FUNCTION_BLOCK SS5b_ps_Ejector (* Composite FB wrapping other FBs *)
  (* Standard: 61499-2 *)
  (* Version 1.0, 2025-08-26, PS_Transformer_for_Unknown *)
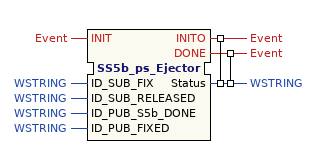
  EVENT_INPUT
    INIT; (* Initialization Request *)
  END_EVENT
  EVENT_OUTPUT
    INITO WITH Status; (* Initialization Confirm *)
    DONE WITH Status; (* Execution Confirmation *)
  END_EVENT
  VAR_INPUT
    ID_SUB_FIX : WSTRING;
    ID_SUB_RELEASED : WSTRING;
    ID_PUB_S5b_DONE : WSTRING;
    ID_PUB_FIXED : WSTRING;
  END_VAR
  VAR_OUTPUT
    Status : WSTRING; (* Output event qualifier *)
  END_VAR
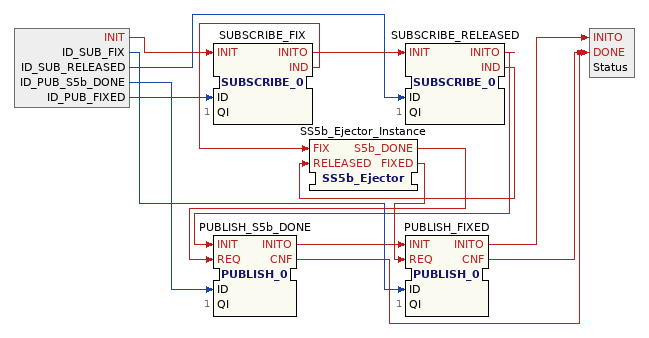
  FBS
    SS5b_Ejector_Instance : SS5b_Ejector;
    SUBSCRIBE_FIX : SUBSCRIBE_0(QI := 1);
    SUBSCRIBE_RELEASED : SUBSCRIBE_0(QI := 1);
    PUBLISH_S5b_DONE : PUBLISH_0(QI := 1);
    PUBLISH_FIXED : PUBLISH_0(QI := 1);
  END_FBS
  EVENT_CONNECTIONS
    INIT TO SUBSCRIBE_FIX.INIT;
    SUBSCRIBE_FIX.INITO TO SUBSCRIBE_RELEASED.INIT;
    SUBSCRIBE_RELEASED.INITO TO PUBLISH_S5b_DONE.INIT;
    PUBLISH_S5b_DONE.INITO TO PUBLISH_FIXED.INIT;
    PUBLISH_FIXED.INITO TO INITO;
    SUBSCRIBE_FIX.IND TO SS5b_Ejector_Instance.FIX;
    SUBSCRIBE_RELEASED.IND TO SS5b_Ejector_Instance.RELEASED;
    SS5b_Ejector_Instance.S5b_DONE TO PUBLISH_S5b_DONE.REQ;
    SS5b_Ejector_Instance.FIXED TO PUBLISH_FIXED.REQ;
    PUBLISH_S5b_DONE.CNF TO DONE;
    PUBLISH_FIXED.CNF TO DONE;
  END_CONNECTIONS
  DATA_CONNECTIONS
    ID_SUB_FIX TO SUBSCRIBE_FIX.ID;
    ID_SUB_RELEASED TO SUBSCRIBE_RELEASED.ID;
    ID_PUB_S5b_DONE TO PUBLISH_S5b_DONE.ID;
    ID_PUB_FIXED TO PUBLISH_FIXED.ID;
  END_CONNECTIONS
END_FUNCTION_BLOCK
